(* This is an empty testsuite with no test cases, so that we can verify that the system still prints the
   test results. *)
FUNCTION_BLOCK FB_EmptyTestSuite EXTENDS TcUnit.FB_TestSuite

END_FUNCTION_BLOCK

(* stored: Version 1.1.0.1, ProductVersion 3.1.4022.18
   POU FB_EmptyTestSuite: Id {1ac34d34-5767-43bd-8deb-b4e9cf217e56}, SpecialFunc None *)
